PROGRAM P50_RecipeControl
VAR
	nRcpIndex		: INT;
	eRecipeRun		: E_RecipeRun ; //레시피 상태
	fbAnalogDeviceRampControl : FB_AnalogDeviceRampControl;
	fbRecipeAnalogInputControlSequencer: FB_RecipeAnalogControlInputSequencer;
	fbOnlyPVUpdate: FB_OnlyPVUpdate;
	fbValveControl: FB_ValveControl;
	
	Pause_TON		: TON;
	Ramp_TON		: FB_TON_Pausable;
	Hold_TON		: FB_TON_Pausable;
	
	loopCount		: ARRAY[1..100] OF INT;
	i				: INT;
END_VAR
VAR CONSTANT
	Pause_MAX		: TIME := T#1800S;
END_VAR

CASE RCP.cmd_RcpOperation OF
	0: //Init State
 		f_ResetTimersAndRCPTimes(fbPause_TON := Pause_TON, fbRamp_TON := Ramp_TON, fbHold_TON := Hold_TON);
		
		FOR i:=1 TO Rcp.iRcpTotalStep DO
			loopCount[i] := Rcp.aRecipe[i].iRecipe[5];
		END_FOR
		
		nRcpIndex := 0;
		Rcp.userState := 0;
		eRecipeRun := E_RecipeRun.Initial;
		GVL_IO.nCaseSignalTower := 5; // White - Idle

	10: //RUN
		IF nRcpIndex = 0 THEN
			nRcpIndex := 1;
		END_IF
		fbAnalogDeviceRampControl();
						
		// CASE 문을 이용한 상태 머신 구현
		CASE eRecipeRun OF
			E_RecipeRun.Initial:
				f_ResetTimersAndRCPTimes(fbPause_TON := Pause_TON, fbRamp_TON := Ramp_TON, fbHold_TON := Hold_TON);
				fbRecipeAnalogInputControlSequencer(rRecipe := RCP.aRecipe[nRcpIndex].rRecipe, rampTime:= TO_UINT(RCP.aRecipe[nRcpIndex].iRecipe[2]));
				fbValveControl(valveSetting:= RCP.aRecipe[nRcpIndex].dRecipe);
				Rcp.userState := 10;// Recipe Running
				GVL_IO.nCaseSignalTower := 3;
				eRecipeRun := E_RecipeRun.Ramp;
				
			E_RecipeRun.Ramp: // Ramp 수행
				Ramp_TON(IN:=TRUE, PT:= RCP.aRecipe[nRcpIndex].iRecipe[2] * T#1S, ET=>RCP.RecipeRunET.ET);
				RCP.RecipeRunET.Mode := E_RecipeRunETMode.Ramp;
				IF Ramp_TON.Q THEN
					Ramp_TON(IN:=FALSE);
					eRecipeRun := E_RecipeRun.CheckHoldTemp;
				END_IF				
				
			E_RecipeRun.CheckHoldTemp: //Hold Temp 확인
				IF RCP.aRecipe[nRcpIndex].cTemp = 0.0 THEN
					Hold_TON(IN:=TRUE, PT:= RCP.aRecipe[nRcpIndex].iRecipe[3] * T#1S, ET=>RCP.RecipeRunET.ET);
					RCP.RecipeRunET.Mode := E_RecipeRunETMode.Hold;
					IF Hold_TON.Q THEN
						Hold_TON(IN:=FALSE);
						eRecipeRun := E_RecipeRun.End; // 레시피 첫 Column 실행
					END_IF
				ELSIF GVL_IO.aController_PV[E_aAnalogInputIO_Index.E_PV_Susceptor_Temp] < RCP.aRecipe[nRcpIndex].cTemp THEN //서셉터 온도가 Wait 온도보다 낮을 때
					Hold_TON(IN:=FALSE);
					eRecipeRun := E_RecipeRun.End; // 레시피 첫 Column 실행
				ELSE // 서셉터 온도가 Wait 온도보다 높을 때
					;// 떨어질 때까지 기다림
				END_IF
				
			E_RecipeRun.End: // 다음 Step 이동 (루프 마지막 단계일 경우, 다음 Step 이동 또는 루프 처음단계로 점프)
				loopCount[nRcpIndex] := loopCount[nRcpIndex] - 1;
				nRcpIndex := nRcpIndex + 1 - (RCP.aRecipe[nRcpIndex].iRecipe[4]) * MIN(loopCount[nRcpIndex], 1);
				IF nRcpIndex > Rcp.iRcpTotalStep THEN
					RCP.cmd_RcpOperation := 50;
				END_IF
				eRecipeRun := E_RecipeRun.Initial;
		END_CASE
		
	20: //PAUSE
		CASE eRecipeRun OF
			E_RecipeRun.Ramp:
				Ramp_TON(PAUSE:=TRUE);		
			E_RecipeRun.CheckHoldTemp:
				Hold_TON(PAUSE:=TRUE);
		END_CASE
		fbOnlyPVUpdate();
		
		Pause_TON(IN:=TRUE, PT:= Pause_MAX, ET=>RCP.Pause_ET); //최대 홀드 시간이 지나면 다음 스텝으로 넘거감
		IF Pause_TON.Q THEN
			Pause_TON(IN:=FALSE);
			eRecipeRun := E_RecipeRun.End; // 레시피 첫 Column 실행
		END_IF

		Rcp.userState := 20;
		GVL_IO.nCaseSignalTower := 5;
		
	30: //RESTART
		Pause_TON(IN:=FALSE);
		CASE eRecipeRun OF
			E_RecipeRun.Ramp:
				Ramp_TON(PAUSE:=FALSE);
			
			E_RecipeRun.CheckHoldTemp:
				Hold_TON(PAUSE:=FALSE);
		END_CASE

		RCP.Pause_ET := T#0S;
		Rcp.userState := 10;
		RCP.cmd_RcpOperation := 10;	
		GVL_IO.nCaseSignalTower := 3;
		
	40: //STOP
		f_ResetTimersAndRCPTimes(fbPause_TON := Pause_TON, fbRamp_TON := Ramp_TON, fbHold_TON := Hold_TON);
		F_StopAnalogRamping_ForRecipe();
		Rcp.userState := 40;
		GVL_IO.nCaseSignalTower := 5;
		
	50: //END
		f_ResetTimersAndRCPTimes(fbPause_TON := Pause_TON, fbRamp_TON := Ramp_TON, fbHold_TON := Hold_TON);
		Rcp.userState := 50;
		fbAnalogDeviceRampControl();
		GVL_IO.nCaseSignalTower := 5;
		
	60: //SKIP
		IF E_RecipeRun.Ramp <= eRecipeRun  AND  eRecipeRun <= E_RecipeRun.CheckHoldTemp THEN
			eRecipeRun := E_RecipeRun.End;
		END_IF
		Rcp.cmd_RcpOperation := 10;
		RCP.Pause_ET := T#0S;
END_CASE
RCP.iRcpStepN := nRcpIndex;

END_PROGRAM

(* stored: Version 1.1.0.1, ProductVersion 3.1.4024.15
   POU P50_RecipeControl: Id {e332a806-fd31-4290-a7c3-27f42c11d38e}, SpecialFunc None *)
